TYPE
	NW_BUF_LONG  : ARRAY[0..NETWORK_BUFFER_LONG_SIZE] OF BYTE;
END_TYPE

(* stored: Version 1.1.0.1, ProductVersion 3.1.4022.7
   DUT NW_BUF_LONG: Id {c232f67b-932e-4a6d-a7c2-44c6a0c2b51d} *)
